PROGRAM motor_PRG
VAR
	motor1_fb :motorFB;
	motor2_FB: motorFB;
END_VAR

// note: this text did not pass the execution check against the stored diagram
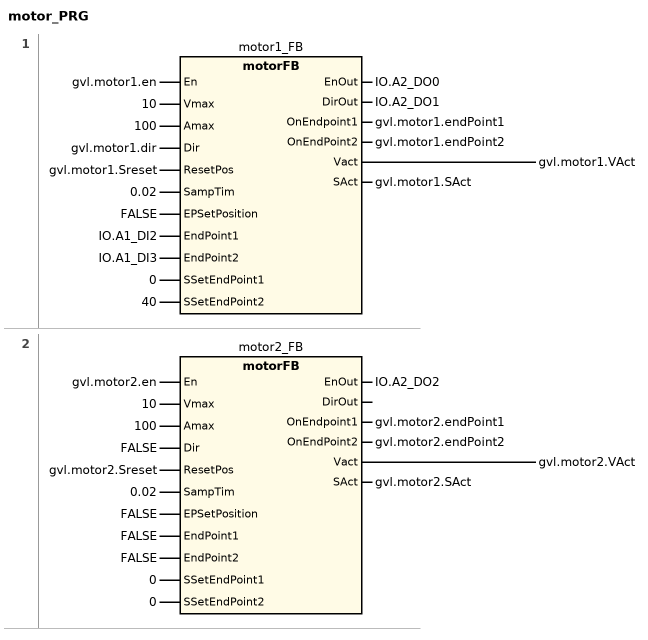
// NETWORK 1
motor1_FB(
    En := gvl.motor1.en,
    Vmax := 10,
    Amax := 100,
    Dir := gvl.motor1.dir,
    ResetPos := gvl.motor1.Sreset,
    SampTim := 0.02,
    EPSetPosition := FALSE,
    EndPoint1 := IO.A1_DI2,
    EndPoint2 := IO.A1_DI3,
    SSetEndPoint1 := 0,
    SSetEndPoint2 := 40,
    EnOut => IO.A2_DO0,
    DirOut => IO.A2_DO1,
    OnEndpoint1 => gvl.motor1.endPoint1,
    OnEndPoint2 => gvl.motor1.endPoint2,
    SAct => gvl.motor1.SAct); // motorFB
gvl.motor1.VAct := motor1_FB.Vact;

// NETWORK 2
motor2_FB(
    En := gvl.motor2.en,
    Vmax := 10,
    Amax := 100,
    Dir := FALSE,
    ResetPos := gvl.motor2.Sreset,
    SampTim := 0.02,
    EPSetPosition := FALSE,
    EndPoint1 := FALSE,
    EndPoint2 := FALSE,
    SSetEndPoint1 := 0,
    SSetEndPoint2 := 0,
    EnOut => IO.A2_DO2,
    OnEndpoint1 => gvl.motor2.endPoint1,
    OnEndPoint2 => gvl.motor2.endPoint2,
    SAct => gvl.motor2.SAct); // motorFB
gvl.motor2.VAct := motor2_FB.Vact;

END_PROGRAM

(* stored: Version 1.1.0.1, ProductVersion 3.1.4024.12
   POU motor_PRG: Id {20c9d9a3-169a-4e39-88de-a798c0e108a8}, SpecialFunc None *)
